DATA_BLOCK "DB_MAP"
{ S7_Optimized_Access := 'FALSE' }
VERSION : 0.1
NON_RETAIN
   STRUCT
      HMI_Word_spare : DWord;
      HMI_Whouse_TRN { S7_SetPoint := 'False'} : "UDT_HMI_Whouse";
      HMI_Whouse_POL { S7_SetPoint := 'False'} : "UDT_HMI_Whouse";
      HMI_Whouse_BUL { S7_SetPoint := 'False'} : "UDT_HMI_Whouse";
      HMI_Whouse_MOL { S7_SetPoint := 'False'} : "UDT_HMI_Whouse";
      HMI_TRN_SmalTank { S7_SetPoint := 'False'} : Array[1..3] of "UDT_HMI_SmallTank";
      HMI_POL_SmalTank { S7_SetPoint := 'False'} : Array[1..10] of "UDT_HMI_SmallTank";
      HMI_BUL_SmalTank { S7_SetPoint := 'False'} : Array[1..4] of "UDT_HMI_SmallTank";
      HMI_MOL_SmalTank { S7_SetPoint := 'False'} : Array[1..12] of "UDT_HMI_SmallTank";
      Scale_CS_1 : "UDT_Siwarex_Core";
      Scale_CS_2 : "UDT_Siwarex_Core";
   END_STRUCT;


BEGIN

END_DATA_BLOCK

